(*Variablen ][ variables*)
usiOldCmdCount := SHR(UINT_TO_USINT(SHL(Axis.DrvToPlc.StateVar,4)),4);
uiCState := SHR(Axis.DrvToPlc.StateVar, 8);

(*Flankenerkennung am Execute Eingang*)
(*Edge detection on Execute input*)
rTrig(CLK:=Execute);
IF rTrig.Q AND uiCState = 16#08 AND NOT Axis.CommandRunning THEN (*Start command*)
	Axis.CommandRunning := TRUE;
	Busy := TRUE;
	uiFbState := 1;
ELSIF rTrig.Q AND Busy THEN (*Restart command / New rising edge on execute input*)
	Axis.CommandRunning := TRUE;
	Busy := TRUE;
	uiFbState := 1;
ELSIF rTrig.Q AND uiCState <> 16#08 THEN (*Axis not ready*)
	uiFbState := 50; (*Error state*)
	Error := TRUE;
	ErrorID := 16#01; (*Axis not ready*)
ELSIF rTrig.Q AND Axis.CommandRunning AND NOT Busy THEN (*Axis already has a command running*)
	uiFbState := 50; (*Error state*)
	Error := TRUE;
	ErrorID := 16#02; (*Axis already has a command running*)
END_IF

IF Busy AND uiCState = 16#04 THEN
	Axis.CommandRunning := FALSE;
	uiFbState := 50;
	Error := TRUE;
	ErrorID := 16#03; (*Axis has error*)
END_IF

IF Busy AND uiCState <> 16#08 THEN
	Axis.CommandRunning := FALSE;
	uiFbState := 50; (*Error state*)
	Error := TRUE;
	ErrorID := 16#04; (*Command interupted*)
ELSIF Busy AND Axis.CommandAborted THEN
	uiFbState := 50; (*Error state*)
	Error := TRUE;
	ErrorID := 16#05; (*Command aborted*)
END_IF

(*State machine*)
CASE uiFbState OF
    0:  ;
        
    1:  (*Check inputs on valid value*)
        IF (-2147483648 < Distance AND Distance < 2147483647)
            AND (0.0 < Velocity)
            AND (0.0 < Acceleration)
            AND (0.0 < Deceleration)
            AND (0.0 < Jerk AND Jerk <= 1600000000)
        THEN
        (*Befehlskopf mit CMD Count berechen und senden ][ Calculate and send command header*)
            usiNewCmdCount := (usiOldCmdCount + 1) MOD 16; (*Command counter MOD 16*)
            Axis.PlcToDrv.MCHeader := 16#0000; (*Reset Header*)
            Axis.PlcToDrv.MCHeader := uiCmdHeader + usiNewCmdCount;
                      
			udiTmpDWord := DINT_TO_UDINT(Distance); (*Position increment*)
            Axis.PlcToDrv.MCParaWord0 := UDINT_TO_UINT(udiTmpDWord);
            Axis.PlcToDrv.MCParaWord1 := UDINT_TO_UINT(ROR(udiTmpDWord, 16));
            
            udiTmpDWord := DINT_TO_UDINT(REAL_TO_DINT(Velocity / 10)); (*Velocity*)
            Axis.PlcToDrv.MCParaWord2 := UDINT_TO_UINT(udiTmpDWord);
            Axis.PlcToDrv.MCParaWord3 := UDINT_TO_UINT(ROR(udiTmpDWord, 16));
            
            udiTmpDWord := DINT_TO_UDINT(REAL_TO_DINT(Acceleration / 100)); (*Acceleration*)
            Axis.PlcToDrv.MCParaWord4 := UDINT_TO_UINT(udiTmpDWord);
            Axis.PlcToDrv.MCParaWord5 := UDINT_TO_UINT(ROR(udiTmpDWord, 16));
            
            udiTmpDWord := DINT_TO_UDINT(REAL_TO_DINT(Deceleration / 100)); (*Deceleration*)
            Axis.PlcToDrv.MCParaWord6 := UDINT_TO_UINT(udiTmpDWord);
            Axis.PlcToDrv.MCParaWord7 := UDINT_TO_UINT(ROR(udiTmpDWord, 16));
            
            udiTmpDWord := DINT_TO_UDINT(REAL_TO_DINT(Jerk) / 1000); (*Jerk*)
            Axis.PlcToDrv.MCParaWord8 := UDINT_TO_UINT(udiTmpDWord);
            Axis.PlcToDrv.MCParaWord9 := UDINT_TO_UINT(ROR(udiTmpDWord, 16));
			
			LM_UptMCI(Axis);
            
            uiFbState := 2;
        ELSE
            Axis.CommandRunning := FALSE;
            uiFbState := 50; (*Error state*)
            Error := TRUE;
            ErrorID := 16#06; (*Invalid input(s)*)
        END_IF;
        
    2:  (*Prüfen ob Befehl ausgeführt ][ Check if command has been executed*)
        IF usiOldCmdCount = usiNewCmdCount AND uiCState = 16#08 AND Axis.DrvToPlc.StateVar.6 THEN
            Done := TRUE;
            Busy := FALSE;
            Axis.PlcToDrv.MCHeader := 16#0000 + usiNewCmdCount; (*Send no operation*)
            Axis.CommandRunning := FALSE;
            uiFbState := 3;
        END_IF;
        
    3:  IF NOT Execute THEN
            uiFbState := 0;
            Busy := FALSE;
            Done := FALSE;
        END_IF;
        
    50: Error := TRUE;
        Busy := FALSE;
        Done := FALSE;
        IF NOT Execute THEN
            uiFbState := 0;
            Error := FALSE;
            ErrorID := 0;
        END_IF;
        
END_CASE;

END_FUNCTION_BLOCK
